(* IEC 61131-3 sources: plcassist-cli/packages/volt-lsp-iec/test-corpus/pro2193/Device/Plc Logic/Application/99 Library/Function Blocks/Triggers, 4 files *)

(* ---- FallingTriggerFB.fb ---- *)
{attribute 'no_explicit_call' := 'Do not call the body of FallingTriggerFB directly! Use methods like Falling to interact with this FB'}
{attribute 'hide_all_locals'}
FUNCTION_BLOCK FallingTriggerFB
VAR
	f_trig			: Standard.F_TRIG;
END_VAR

END_FUNCTION_BLOCK

// Monitor an input for a falling edge. Use property Q to get edge.
METHOD PUBLIC Call
VAR_INPUT
	CLK	: BOOL;
END_VAR

// Use this method if you need the trigger output more than once per PLC cycle.
f_trig(
	CLK	:= CLK,
	Q   => );
END_METHOD

// Triggers on falling edge of input. !!Only call this method once per PLC Cycle!!
METHOD PUBLIC Falling : BOOL
VAR_INPUT
	CLK	: BOOL;
END_VAR
Call(CLK);
Falling := Q;
END_METHOD

// Rising edge of the input signal
PROPERTY PUBLIC Q : BOOL

// Attribute 'monitoring':='call' is not needed here.
GET
VAR
END_VAR
Q := f_trig.Q;
END_GET
END_PROPERTY

(* ---- RisingTriggerFB.fb ---- *)
{attribute 'no_explicit_call' := 'Do not call the body of RisingTriggerFB directly! Use methods like Rising to interact with this FB'}
{attribute 'hide_all_locals'}
FUNCTION_BLOCK RisingTriggerFB
VAR
	r_trig			: Standard.R_TRIG;
END_VAR

END_FUNCTION_BLOCK

// Monitor an input for a rising edge. Use property Q to get edge.
METHOD PUBLIC Call
VAR_INPUT
	CLK	: BOOL;
END_VAR

// Use this method if you need the trigger output more than once per PLC cycle.
r_trig(
	CLK	:= CLK,
	Q   => );
END_METHOD

// Triggers on rising edge of input. !!Only call this method once per PLC Cycle!!
METHOD PUBLIC Rising : BOOL
VAR_INPUT
	CLK	: BOOL;
END_VAR
Call(CLK);
Rising := Q;
END_METHOD

// Rising edge of the input signal
PROPERTY PUBLIC Q : BOOL

// Attribute 'monitoring':='call' is not needed here.
GET
VAR
END_VAR
Q := r_trig.Q;
END_GET
END_PROPERTY

(* ---- TriggerFB.fb ---- *)
// Rising / Falling trigger FB, with separate outputs for rising and falling trigger
{attribute 'no_explicit_call' := 'Do not call the body of TriggerFB directly! Use methods like Rising to interact with this FB'}
{attribute 'hide_all_locals'}
FUNCTION_BLOCK TriggerFB
VAR
	xRisingEdge		: BOOL;	// The rising edge of the input signal
	xFallingEdge	: BOOL;	// The falling edge of the input signal
	xEdge			: BOOL;	// Memory flag, to detect a change in input
END_VAR

END_FUNCTION_BLOCK

// Triggers on both rising and falling edge of input. !!Only call this method once per PLC Cycle!!
METHOD PUBLIC AnyEdge : BOOL
VAR_INPUT
	CLK	: BOOL;
END_VAR
Call(CLK);
AnyEdge := Q_Rising OR Q_Falling;
END_METHOD

// Monitor an input for a rising and falling edge. Use properties Q_R and Q_F to get edges.
METHOD PUBLIC Call
VAR_INPUT
	CLK	: BOOL;
END_VAR

// Use this method if you need the trigger output more than once per PLC cycle.
xRisingEdge		:= CLK AND NOT xEdge;
xFallingEdge	:= NOT CLK AND xEdge;
xEdge			:= CLK;
END_METHOD

// Triggers on falling edge of input. !!Only call this method once per PLC Cycle!!
METHOD PUBLIC Falling : BOOL
VAR_INPUT
	CLK	: BOOL;
END_VAR
Call(CLK);
Falling := Q_Falling;
END_METHOD

// Triggers on rising edge of input. !!Only call this method once per PLC Cycle!!
METHOD PUBLIC Rising : BOOL
VAR_INPUT
	CLK	: BOOL;
END_VAR
Call(CLK);
Rising := Q_Rising;
END_METHOD

// Falling edge of the input signal
PROPERTY PUBLIC Q_Falling : BOOL
GET
VAR
END_VAR
Q_Falling := xFallingEdge;
END_GET
END_PROPERTY

// Rising edge of the input signal
PROPERTY PUBLIC Q_Rising : BOOL

// Attribute 'monitoring':='call' is not needed here.
GET
VAR
END_VAR
Q_Rising := xRisingEdge;
END_GET
END_PROPERTY

(* ---- TriggerRealFB.fb ---- *)
// monitors a REAL for change
{attribute 'hide_all_locals'}
FUNCTION_BLOCK TriggerRealFB
VAR_INPUT
	IN		: REAL;
	RES		: REAL;
END_VAR
VAR_OUTPUT
	Q		: BOOL;
	D		: REAL;
END_VAR
VAR
	LAST_IN	: REAL;
END_VAR

// this block is similar to the IEC Standard R_trig and F_trig but it monitors a REAL for change.
// if the valiue on IN changes more then D from the last value it will generate trigger and display the difference in output D.
// the trigger will only be active for one cycle.

D := IN - LAST_IN;
Q := ABS(D) > RES;
IF Q THEN
	LAST_IN := IN;
END_IF
D := IN - LAST_IN;

END_FUNCTION_BLOCK
